// TIA Portal V15.1 export
// export: Created 2020-06-12T07:35:49.5224609Z, ExportSetting None, DisplayName Totally Integrated Automation Portal, DisplayVersion V15.1, DisplayName TIA Portal Openness, DisplayVersion V15.1, DisplayName STEP 7 Professional, DisplayVersion V15.1, DisplayName STEP 7 Safety, DisplayVersion V15.1, DisplayName WinCC Advanced, DisplayVersion V15.1
FUNCTION "ContrSlow_call" : Void   // FC184, FBD
TITLE = Slow PID/SM controllers
{ S7_Optimized_Access := 'TRUE' }
// stored: SetENOAutomatically False
BEGIN

REGION Network 1: Cooling water system, base temperature control
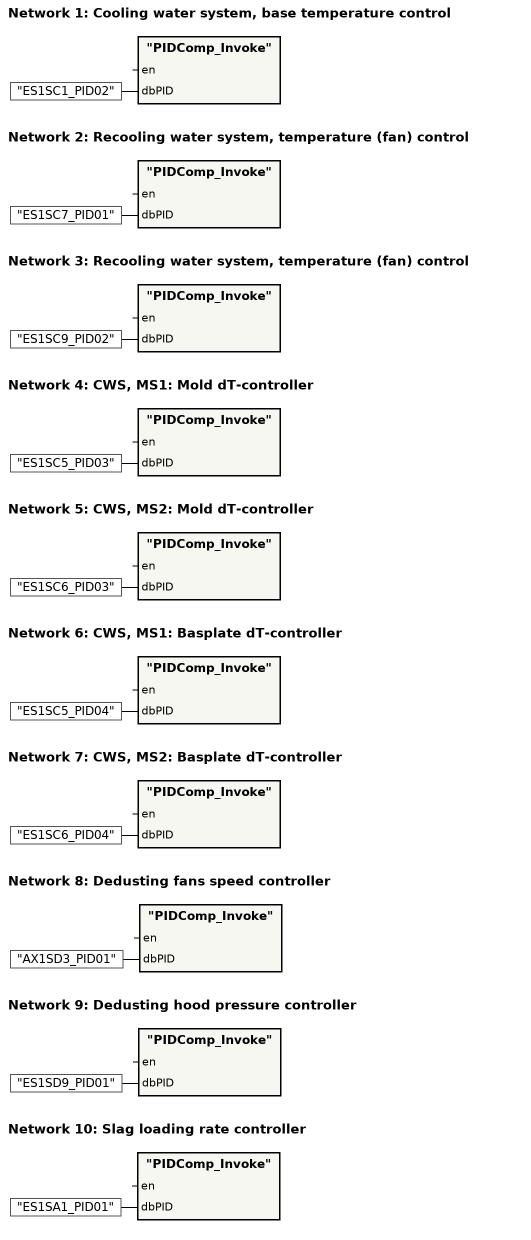
   "PIDComp_Invoke"(dbPID := "ES1SC1_PID02");
END_REGION

REGION Network 2: Recooling water system, temperature (fan) control
   "PIDComp_Invoke"(dbPID := "ES1SC7_PID01");
END_REGION

REGION Network 3: Recooling water system, temperature (fan) control
   "PIDComp_Invoke"(dbPID := "ES1SC9_PID02");
END_REGION

REGION Network 4: CWS, MS1: Mold dT-controller
   "PIDComp_Invoke"(dbPID := "ES1SC5_PID03");
END_REGION

REGION Network 5: CWS, MS2: Mold dT-controller
   "PIDComp_Invoke"(dbPID := "ES1SC6_PID03");
END_REGION

REGION Network 6: CWS, MS1: Basplate dT-controller
   "PIDComp_Invoke"(dbPID := "ES1SC5_PID04");
END_REGION

REGION Network 7: CWS, MS2: Basplate dT-controller
   "PIDComp_Invoke"(dbPID := "ES1SC6_PID04");
END_REGION

REGION Network 8: Dedusting fans speed controller
   "PIDComp_Invoke"(dbPID := "AX1SD3_PID01");
END_REGION

REGION Network 9: Dedusting hood pressure controller
   "PIDComp_Invoke"(dbPID := "ES1SD9_PID01");
END_REGION

REGION Network 10: Slag loading rate controller
   "PIDComp_Invoke"(dbPID := "ES1SA1_PID01");
END_REGION
END_FUNCTION
